// TIA Portal V18 export
DATA_BLOCK "FB10-heater_DB_1"   // DB12
VERSION : 0.1
// stored: AutoNumber true, DBAccessibleFromOPCUA true, InstanceOfName FB10-heater, InstanceOfType FB
"FB10-heater"
   // VAR_INPUT
   //    ON : Bool;
   //    "Temperature oC" : Real;
   //    "Set temperature" : Real;
   //    "pre shutdown temperature" : Real;
   //    "Limit under temperature" : Real;
   //    "Limit Over temperature" : Real;
   //    "heating adjustment hysteresis" : Real;
   //    "Minimum ON time" : Real;
   //    "Minimum OFF time" : Real;
   // END_VAR
   // VAR_OUTPUT
   //    "Heater PWM" : Bool;
   //    "Heater Temperature under Limit" : Bool;
   //    "Heater Temperature Over Limit" : Bool;
   //    "Temperature Above SP" { ExternalAccessible := 'False'; ExternalVisible := 'False'; ExternalWritable := 'False'} : Bool;
   //    "Dispensing Stop undertemperature" { ExternalAccessible := 'False'; ExternalVisible := 'False'; ExternalWritable := 'False'} : Bool;
   // END_VAR
   // VAR
   //    "set temperature after hysteresis" : Real;
   //    "On time in msec" : DInt;
   //    "off time in msec" : DInt;
   //    "On timer triggered" : Bool;
   //    "off time triggered" : Bool;
   //    IEC_Timer_0_Instance { S7_SetPoint := 'True'} : TON_TIME;
   //    IEC_Timer_0_Instance_1 { S7_SetPoint := 'True'} : TON_TIME;
   // END_VAR
BEGIN
END_DATA_BLOCK
